{attribute 'GeneratedUsingTerminal: EL9930-0000-0016'}
{attribute addProperty BoxType "EL9930-0000-0016"}
{attribute addProperty Id "A_0002_EL9930_0001_0016EL9930_07FC3A1D4A_0003_EL9930_0000_0017A_0003_EL9930_0000_0017_96B57C1D4"}
{attribute addProperty CRC "4157294235"}
{attribute addProperty Size "8"}
{attribute addProperty Name "A_0001(EL9930-0000-0016)"}
TYPE A_0001_EL9930_0000_0016_F7CB469B EXTENDS EL9930_77AEBA45 :
STRUCT
	{attribute addProperty Name "A_0002(EL9930-0001-0016)"}
	{attribute addProperty PreviousPort "A_0001(EL9930-0000-0016) : B"}
	A_0002_EL9930_0001_0016 : EL9930_07FC3A1D;
	{attribute addProperty Name "A_0003(EL9930-0000-0017)"}
	{attribute addProperty PreviousPort "A_0002(EL9930-0001-0016) : B"}
	A_0003_EL9930_0000_0017 : A_0003_EL9930_0000_0017_96B57C1D;
END_STRUCT
END_TYPE

(* stored: Version 1.2.0.0, ProductVersion 3.1.4024.11
   DUT A_0001_EL9930_0000_0016_F7CB469B: Id {c7739f9a-bf0b-49d5-82b7-585ddbe48ee9} *)
